TYPE "rxRecordWritePub"
TITLE = Type:"RX record write publisher"
VERSION : 0.1
//["version","date","author","description"],
//["v1.0","2022-10-12","cyanezf","First version"]
//
   STRUCT
      providerStatus : Byte;   // Bit 0: 1=Se ha establecido la comunicación con el otro lado del bus y los módulos "RD READ PUB" y "LOCAL RD READ PUB" se han configurado en el otro lado del bus
   END_STRUCT;

END_TYPE

